//-----------------------------------------------------------------------------------------
//
//                  				ST_Tool_Name
//
//								Structure nom outil 			
//-----------------------------------------------------------------------------------------
//
//Auteur: G.GOETZ (inspired by S.FLEURY)
//Création: 20.01.2026
//Dernière modification : 20.01.2026 (G.GOETZ)
//       			
//-----------------------------------------------------------------------------------------
//
//     							Liste des modifications  	
//
// 20.01.2026 (G.GOETZ) -> Création		
//-----------------------------------------------------------------------------------------

TYPE ST_Tool_Name :
STRUCT
	
	(** SETUP STRING **)
		Name : STRING[GV_Tool_Magazine.iNumCharaToolName] ; // Name
	
END_STRUCT
END_TYPE

(* stored: Version 1.1.0.1, ProductVersion 3.1.4026.17
   DUT ST_Tool_Name: Id {06f1a297-0c58-4a9c-9e13-9613b646fdcb} *)
